% RSLogix 500 project SEALIN_BAK000.RSS, saved by version 8.30.00.16 %
PROJECT "SEALIN"    % processor: Bul.1763 MicroLogix 1100 Series B %

PROGRAM FILES
  LAD 2   2 rungs

DATA FILES
  O0 OUTPUT  4 elements
  I1 INPUT  6 elements
  S2 STATUS  66 elements
  B3 BINARY  1 elements
  T4 TIMER  1 elements
  C5 COUNTER  1 elements
  R6 CONTROL  1 elements
  N7 INTEGER  1 elements
  F8 FLOAT  1 elements

LADDER 2
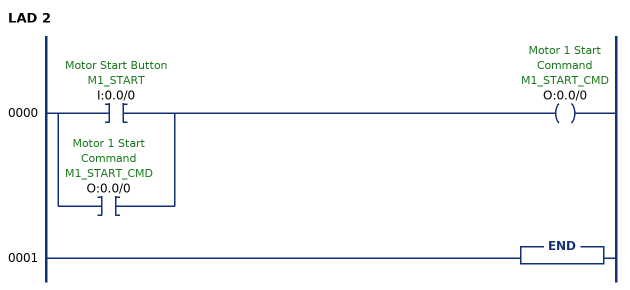
% Rung: 0 %  % edit flag set %
SOR BST XIC I:0.0/0 NXB XIC O:0.0/0 BND OTE O:0.0/0 EOR
%   I:0.0/0  M1_START  "Motor Start Button" %
%   O:0.0/0  M1_START_CMD  "Motor 1 Start Command" %
% Rung: 1 %
SOR END EOR
